{attribute 'qualified_only'}
{attribute 'strict'}
{attribute 'to_string'}
TYPE E_MESSAGE_CHECK :
(
  // 9000 --> here comes your error
  MSG_CHECK_INVALID_POINTER             := 9000,
  MSG_CHECK_INVALID_POINTER_TIME,
  MSG_CHECK_INVALID_POINTER_LIST,
  MSG_CHECK_INVALID_POINTER_MSG_IDX,
  MSG_CHECK_INVALID_POINTER_ERR_IDX,
  MSG_CHECK_INVALID_POINTER_ROOT_FILE,
  MSG_CHECK_INVALID_POINTER_ROOT_DIR,
  MSG_CHECK_INVALID_POINTER_CTRL,
  MSG_CHECK_INVALID_POINTER_STATE,

  // 10000 --> here comes your man
  MSG_CHECK_DONE                        := 10000
)UINT;
END_TYPE

(* stored: Version 1.1.0.1, ProductVersion 3.1.4026.13
   DUT E_MESSAGE_CHECK: Id {56cd86e7-f2ee-489b-81d6-76ce6e9d72dc} *)
